// TIA Portal V17 export
// export: Created 2025-03-05T08:03:01.2107892Z, ExportSetting WithDefaults, DisplayName Totally Integrated Automation Portal, DisplayVersion V17 Update 8, DisplayName TIA Portal Openness, DisplayVersion V17 Update 8, DisplayName TIA Portal Version Control Interface, DisplayVersion V17, DisplayName SINAMICS Startdrive Advanced, DisplayVersion V17 SP2, DisplayName SINAMICS Startdrive G110M, G120, G120C, G120D, G120P, G115D, DisplayVersion V17 SP2, DisplayName SINAMICS Startdrive G130, G150, S120, S150, SINAMICS MV, S210, DisplayVersion V17 SP2, DisplayName STEP 7 Professional, DisplayVersion V17 Update 8, DisplayName SINUMERIK ONE STEP 7 Toolbox, DisplayVersion V17 Update 12, DisplayName SINUMERIK 840D sl STEP 7 Toolbox, DisplayVersion V17 Update 12, DisplayName STEP 7 Safety, DisplayVersion V17 Update 6, DisplayName WinCC Advanced, DisplayVersion V17 Update 8
FUNCTION "FC21000_POWDER_FEEDER_MAIN" : Void   // FC21000, LAD
TITLE = FC21000 POWDER FEEDER MAIN
{ S7_Optimized_Access := 'TRUE' }
VERSION : 0.1
// stored: AutoNumber false, IsIECCheckEnabled false, SetENOAutomatically false, UDAEnableTagReadback false
   VAR_TEMP
      ret_val_1 : Int;
      OPTIONS_OFF : Bool;
      OPTIONS_ON : Bool;
      POWDER_SWITCH_OPTION : Bool;
      MEDICOAT_OPTION : Bool;
   END_VAR
BEGIN

REGION Network 1: OPTIONS OFF
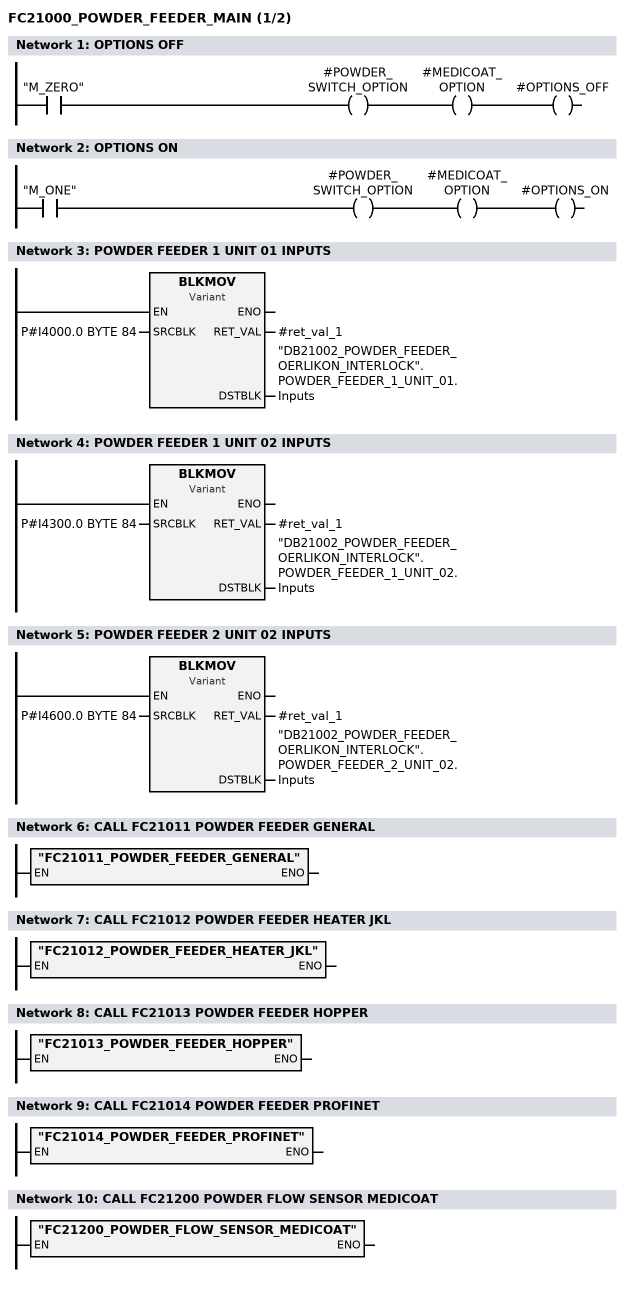
   RUNG wire#powerrail
      Contact( "M_ZERO" )
      Coil( #POWDER_SWITCH_OPTION )
      Coil( #MEDICOAT_OPTION )
      Coil( #OPTIONS_OFF )
   END_RUNG
   // the same network as SCL:
   #POWDER_SWITCH_OPTION := "M_ZERO";
   #MEDICOAT_OPTION := "M_ZERO";
   #OPTIONS_OFF := "M_ZERO";
END_REGION

REGION Network 2: OPTIONS ON
   RUNG wire#powerrail
      Contact( "M_ONE" )
      Coil( #POWDER_SWITCH_OPTION )
      Coil( #MEDICOAT_OPTION )
      Coil( #OPTIONS_ON )
   END_RUNG
   // the same network as SCL:
   #POWDER_SWITCH_OPTION := "M_ONE";
   #MEDICOAT_OPTION := "M_ONE";
   #OPTIONS_ON := "M_ONE";
END_REGION

REGION Network 3: POWDER FEEDER 1 UNIT 01 INPUTS
   RUNG wire#powerrail
      { S7_Templates := "blk_type := Variant" } BLKMOV(SRCBLK := P#I4000.0 BYTE 84, RET_VAL => #ret_val_1, DSTBLK => "DB21002_POWDER_FEEDER_OERLIKON_INTERLOCK".POWDER_FEEDER_1_UNIT_01.Inputs)
   END_RUNG
   // the same network as SCL:
   #ret_val_1 := BLKMOV(SRCBLK := P#I4000.0 BYTE 84,
                        DSTBLK => "DB21002_POWDER_FEEDER_OERLIKON_INTERLOCK".POWDER_FEEDER_1_UNIT_01.Inputs);
END_REGION

REGION Network 4: POWDER FEEDER 1 UNIT 02 INPUTS
   RUNG wire#powerrail
      { S7_Templates := "blk_type := Variant" } BLKMOV(SRCBLK := P#I4300.0 BYTE 84, RET_VAL => #ret_val_1, DSTBLK => "DB21002_POWDER_FEEDER_OERLIKON_INTERLOCK".POWDER_FEEDER_1_UNIT_02.Inputs)
   END_RUNG
   // the same network as SCL:
   #ret_val_1 := BLKMOV(SRCBLK := P#I4300.0 BYTE 84,
                        DSTBLK => "DB21002_POWDER_FEEDER_OERLIKON_INTERLOCK".POWDER_FEEDER_1_UNIT_02.Inputs);
END_REGION

REGION Network 5: POWDER FEEDER 2 UNIT 02 INPUTS
   RUNG wire#powerrail
      { S7_Templates := "blk_type := Variant" } BLKMOV(SRCBLK := P#I4600.0 BYTE 84, RET_VAL => #ret_val_1, DSTBLK => "DB21002_POWDER_FEEDER_OERLIKON_INTERLOCK".POWDER_FEEDER_2_UNIT_02.Inputs)
   END_RUNG
   // the same network as SCL:
   #ret_val_1 := BLKMOV(SRCBLK := P#I4600.0 BYTE 84,
                        DSTBLK => "DB21002_POWDER_FEEDER_OERLIKON_INTERLOCK".POWDER_FEEDER_2_UNIT_02.Inputs);
END_REGION

REGION Network 6: CALL FC21011 POWDER FEEDER GENERAL
   RUNG wire#powerrail
      "FC21011_POWDER_FEEDER_GENERAL"()
   END_RUNG
   // the same network as SCL:
   "FC21011_POWDER_FEEDER_GENERAL"();
END_REGION

REGION Network 7: CALL FC21012 POWDER FEEDER HEATER JKL
   RUNG wire#powerrail
      "FC21012_POWDER_FEEDER_HEATER_JKL"()
   END_RUNG
   // the same network as SCL:
   "FC21012_POWDER_FEEDER_HEATER_JKL"();
END_REGION

REGION Network 8: CALL FC21013 POWDER FEEDER HOPPER
   RUNG wire#powerrail
      "FC21013_POWDER_FEEDER_HOPPER"()
   END_RUNG
   // the same network as SCL:
   "FC21013_POWDER_FEEDER_HOPPER"();
END_REGION

REGION Network 9: CALL FC21014 POWDER FEEDER PROFINET
   RUNG wire#powerrail
      "FC21014_POWDER_FEEDER_PROFINET"()
   END_RUNG
   // the same network as SCL:
   "FC21014_POWDER_FEEDER_PROFINET"();
END_REGION

REGION Network 10: CALL FC21200 POWDER FLOW SENSOR MEDICOAT
   RUNG wire#powerrail
      "FC21200_POWDER_FLOW_SENSOR_MEDICOAT"()
   END_RUNG
   // the same network as SCL:
   "FC21200_POWDER_FLOW_SENSOR_MEDICOAT"();
END_REGION

REGION Network 11: POWDER FEEDER 1 UNIT 01 OUTPUTS
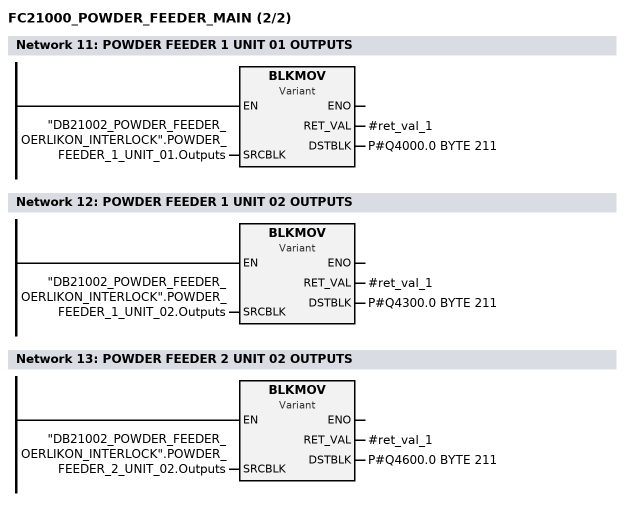
   RUNG wire#powerrail
      { S7_Templates := "blk_type := Variant" } BLKMOV(SRCBLK := "DB21002_POWDER_FEEDER_OERLIKON_INTERLOCK".POWDER_FEEDER_1_UNIT_01.Outputs, RET_VAL => #ret_val_1, DSTBLK => P#Q4000.0 BYTE 211)
   END_RUNG
   // the same network as SCL:
   #ret_val_1 := BLKMOV(SRCBLK := "DB21002_POWDER_FEEDER_OERLIKON_INTERLOCK".POWDER_FEEDER_1_UNIT_01.Outputs,
                        DSTBLK => P#Q4000.0 BYTE 211);
END_REGION

REGION Network 12: POWDER FEEDER 1 UNIT 02 OUTPUTS
   RUNG wire#powerrail
      { S7_Templates := "blk_type := Variant" } BLKMOV(SRCBLK := "DB21002_POWDER_FEEDER_OERLIKON_INTERLOCK".POWDER_FEEDER_1_UNIT_02.Outputs, RET_VAL => #ret_val_1, DSTBLK => P#Q4300.0 BYTE 211)
   END_RUNG
   // the same network as SCL:
   #ret_val_1 := BLKMOV(SRCBLK := "DB21002_POWDER_FEEDER_OERLIKON_INTERLOCK".POWDER_FEEDER_1_UNIT_02.Outputs,
                        DSTBLK => P#Q4300.0 BYTE 211);
END_REGION

REGION Network 13: POWDER FEEDER 2 UNIT 02 OUTPUTS
   RUNG wire#powerrail
      { S7_Templates := "blk_type := Variant" } BLKMOV(SRCBLK := "DB21002_POWDER_FEEDER_OERLIKON_INTERLOCK".POWDER_FEEDER_2_UNIT_02.Outputs, RET_VAL => #ret_val_1, DSTBLK => P#Q4600.0 BYTE 211)
   END_RUNG
   // the same network as SCL:
   #ret_val_1 := BLKMOV(SRCBLK := "DB21002_POWDER_FEEDER_OERLIKON_INTERLOCK".POWDER_FEEDER_2_UNIT_02.Outputs,
                        DSTBLK => P#Q4600.0 BYTE 211);
END_REGION
END_FUNCTION
